# B&R Automation Studio project OpcUaSample410_BrbLibUa103 (part 16)

#### Set_BrbUaSrvGetMethodOperateText.c - Test set
```c
#include <bur/plctypes.h>

#ifdef _DEFAULT_INCLUDES
#include <AsDefault.h>
#endif

#include "UnitTest.h"
#include "BrbAsserts.h"
#include <string.h>

// NOLINTBEGIN(readability-*, bugprone-easily-swappable-parameters, bugprone-branch-clone, clang-diagnostic-invalid-utf8, clang-diagnostic-invalid-source-encoding, clang-diagnostic-pointer-arith, clang-diagnostic-strict-prototypes, clang-diagnostic-bad-function-cast, clang-analyzer-security.insecureAPI.*, hicpp-uppercase-literal-suffix, cppcoreguidelines-*, performance-*)
_TEST BrbUaSrvGetMethodOperateText_NulPtr(void)
{
	dwordOut = BrbUaSrvGetMethodOperateText(0, 0, 0);
	TEST_ASSERT_EQUAL_INT(0x80460000, dwordOut); // = Bad_StructureMissing

	// Finished
	TEST_DONE;
}

_TEST BrbUaSrvGetMethodOperateText_Get(void)
{
	methodOperationAction = UaMoa_CheckIsCalled;
	dwordOut = BrbUaSrvGetMethodOperateText(methodOperationAction, stringIn0, sizeof(stringIn0));
	TEST_ASSERT_EQUAL_INT(0x00000000, dwordOut); // = Good
	TEST_ASSERT_EQUAL_STRING("CheckIsCalled", stringIn0);

	methodOperationAction = UaMoa_Finished;
	dwordOut = BrbUaSrvGetMethodOperateText(methodOperationAction, stringIn0, sizeof(stringIn0));
	TEST_ASSERT_EQUAL_INT(0x00000000, dwordOut); // = Good
	TEST_ASSERT_EQUAL_STRING("Finished", stringIn0);

	// Finished
	TEST_DONE;
}

// NOLINTEND(readability-*, bugprone-easily-swappable-parameters, bugprone-branch-clone, clang-diagnostic-invalid-utf8, clang-diagnostic-invalid-source-encoding, clang-diagnostic-pointer-arith, clang-diagnostic-strict-prototypes, clang-diagnostic-bad-function-cast, clang-analyzer-security.insecureAPI.*, hicpp-uppercase-literal-suffix, cppcoreguidelines-*, performance-*)

/*
B+R UnitTest: This is generated code.
Do not edit! Do not move!
Description: UnitTest Testprogramm infrastructure (TestSet).
LastUpdated: 2023-04-25 13:44:36Z
By B+R UnitTest Helper Version: 2.0.1.59
*/
UNITTEST_FIXTURES(fixtures)
{
	new_TestFixture("BrbUaSrvGetMethodOperateText_NulPtr", BrbUaSrvGetMethodOperateText_NulPtr),
	new_TestFixture("BrbUaSrvGetMethodOperateText_Get", BrbUaSrvGetMethodOperateText_Get),
};

UNITTEST_CALLER_COMPLETE_EXPLICIT(Set_BrbUaSrvGetMethodOperateText, "Set_BrbUaSrvGetMethodOperateText", 0, 0, fixtures, 0, 0, 0);
```

### Package Logical/Tasks/Template - Muster für einen Task

### ReadMe.txt
```
Das ist nur ein Muster, um damit schnell die Grund-Struktur eines neuen Tasks zu erstellen.
Es wird für das Beispiel nicht benötigt.
```

### Program Logical/Tasks/Template/TemplateC/TemplateC (ANSIC) - Muster für einen C-Task

#### TemplateC.c - Implementation code
```c
#include <bur/plctypes.h>

#ifdef _DEFAULT_INCLUDES
	#include <AsDefault.h>
#endif

// NOLINTBEGIN(readability-*, bugprone-easily-swappable-parameters, bugprone-branch-clone, clang-diagnostic-invalid-utf8, clang-diagnostic-invalid-source-encoding, clang-diagnostic-pointer-arith, clang-diagnostic-strict-prototypes, clang-diagnostic-shadow, clang-diagnostic-bad-function-cast, clang-analyzer-security.insecureAPI.*, hicpp-uppercase-literal-suffix, hicpp-function-size, cppcoreguidelines-*, performance-*)

void _INIT Init(void)
{
}

void _CYCLIC Cyclic(void)
{
}

void _EXIT Exit(void)
{
}

// NOLINTEND(readability-*, bugprone-easily-swappable-parameters, bugprone-branch-clone, clang-diagnostic-invalid-utf8, clang-diagnostic-invalid-source-encoding, clang-diagnostic-pointer-arith, clang-diagnostic-strict-prototypes, clang-diagnostic-shadow, clang-diagnostic-bad-function-cast, clang-analyzer-security.insecureAPI.*, hicpp-uppercase-literal-suffix, hicpp-function-size, cppcoreguidelines-*, performance-*)
```

### Program Logical/Tasks/Template/TemplateST/TemplateST (IEC) - Muster für einen ST-Task

#### TemplateST.st - Init, cyclic, exit code
```iecst
PROGRAM _INIT
END_PROGRAM

PROGRAM _CYCLIC
END_PROGRAM

PROGRAM _EXIT
END_PROGRAM
```

### Package Logical/Tasks/ServerData - Daten für den eigenen OpcUa-Server

### ReadMe.txt
```
Hier werden Variablen zur Verfügung gestellt, die der eigene OpcUa-Server veröffentlicht.

Der Server ist in der System-Konfiguration unter 'OPCUA Server' parametriert. Es ist das PV-Informationsmodell V2.0
eingestellt.

Die User-/Roles-Parametrierung ist unter ConfigurationView/AccessAndSecurity/UserRoleSystem.  Hier ist folgende
Authentifizierung angegeben:
	Username:			Admin
	Password:			admin

Daten sind als globale Variable 'gVarsGlobal' und als lokale Variable 'VarsLocal' angelegt.
Sie wurden in der Datei 'OpcUaMap.uad' (siehe ConfigurationView/Connectivity/OpcUa) für den Server konfiguriert.
Sie enthalten die Strukturen 'Read', 'Write' und 'ReadWrite', welche auch so parametriert sind.
Diese wiederum enthalten jeweils ein Unterelement jeden Standard-Datentyps.
Definition siehe LogicalView/Global.typ.
Die Elemente der Unter-Struktur 'Read' werden im Task-Takt (500ms) geändert.

Eine Übersetzung des Attributes 'Description' ist beispielhaft bei den beiden Knoten 'gVarsGlobal' und 'VarsLocal'
implementiert. Dabei werden die Texte aus der Datei 'Texts/OpcUaServerTexts' verwendet.

Ausserdem gibt es die Strukturen 'WriteC' und 'WriteST', auf deren Elemente teilweise von den Clients geschrieben wird.

Einsatz von dynamischen Arrays:
	Auf einer SPS kann ein Array nie dynamisch sein, also keine variable Länge haben. Die Länge eines Arrays
	muss zur Projektierungszeit im AS  festgelegt werden und kann zur Laufzeit nicht mehr geändert werden.
	OpcUa untersützt jedoch dynamische Arrays.
	Der B&R-Server kann mit einem Trick ein in der SPS deklariertes Array OpcUa-seitig als dynamisch
	ausliefern. Auch ein empfangenes dynamisches Array kann so auf ein festes SPS-Array übertragen werden.
	Als einfaches Beispiel dient hier die Variable 'DynamicUintArrayLength', welche durch einen selbstdefinierten
	Datentyp deklariert wird. Der Datentyp sieht so aus:
		DynamicUintArrayLength_TYP : 	STRUCT
			nLength : UAArrayLength;
			anData : ARRAY[0..9]OF UINT;
		END_STRUCT;
	Das Element 'anData' enthält das Array mit fester maximaler Länge, wie auf der SPS benötigt.
	Das Element 'nLength' enthält die Anzahl der gültigen Array-Elemente. Durch Setzen dieses Wertes wird	das am
	OpcUa-Server bediente Array angepasst.
	Die Variable wird ganz normal am OpcUa-Server freigegeben (ohne Unter-Elemente). Das System erkennt aufgrund der
	Deklaration, dass diese	Variable ein dynamisches Array ist und behandelt es entsprechend.
	Bei einem DirectRead oder als MonitoredItem einer Subscription wird ein Array mit der aktuellen Länge übertragen.
	Bei einem DirectWrite werden die als Array übertragene Werte in 'anData' geschrieben und 'nLength' entsprechend
	gesetzt.
	Die Länge kann anstatt als 'UAArrayLength' auch als 'UANoOfElements' deklariert werden. Der Unterschied ist das Format,
	in welchem das Array an den Client übertragen bzw. vom Client erwartet wird:
		UAArrayLength:		Wird als Uint16[] übertragen.
		UANoOfElements:		Wird als ExtensionObject übertragen. Es enthält das UINT-Array.

	Als Beispiel für die zweite Variante ist die Variable 'DynamicUintArrayElements' implementiert. Über einen Test-Client
	wie UaExpert oder RnCommTest kann der Unterschied des Formats sehr leicht erkannt werden.
	Welche Variante verwendet werden sollte, hängt davon ab, mit welchem Format der Client umgehen kann. Sps-seitig ist
	Behandlung identisch.

	Dieses Konzept funktioniert nicht nur mit allen Standard-Datentypen, sondern auch mit Struktur-Arrays. Als Beispiele
	sind die beiden Variablen 'DynamicStructArrayLength' bzw. 'DynamicStructArrayElements' implementiert.
	Achtung: Mindestens eine skalare Instanz der verwendeten Struktur muss freigegeben sein, damit der Datentyp vom Server
	veröffentlicht wird und es dem Client so ermöglicht, die Struktur aufzulösen. Wenn der Struktur-Datentyp nur im Array
	verwendet wird, ist dies nicht der Fall!

	Achtung: Bei einem Schreib-Zugriff auf ein dynamisches Array darf die Anzahl der geschriebenen Elemente NICHT die
	Länge des Array 'anData' überschreiten, da der Server dann die empfangenen Daten nicht in das Array übertragen kann.
	Wird dies	doch gemacht, führt der Server den Schreibauftrag nicht aus und gibt den Status
	'0x8074000' = BadTypeMismatch	zurück!

	Hinweis: Bei dynamischen Arrays werden nur 1-dimensionale, aber keine mehrdimensionalen Arrays unterstützt.

	Implementierung im Beispiel-Task:
	Die Arrays werden im Init des Tasks vorbesetzt. Im zyklischen Teil (500ms) werden nur die Längen der einzelnen
	Instanzen zufällig verändert.

	Bekannte Bugs in AR-Versionen:
	Behoben ab C4.72:
		Definition mit 'UAArrayLength':
			Bei einem dynamischen Standard-Datentypen-Array, welches vom Client über eine	Subscription abonniert wurde,
			lieferte der Server bei einer Wert-Änderung nicht das Array, sondern nur die aktuelle Länge.
			Hinweis: Mit 'UANoOfElements' funktionierte es korrekt.

	Behoben ab B4.73:
		Definition mit 'UAArrayLength':
			Die Verwendung als Methoden-Argument funktioniert nicht korrekt. Werden weniger Elemente als die maximale Anzahl
			an Elementen gesendet, quittiert dies der Server mit '0x80AB000 = BadInvalidArgument'
			Hinweis: Mit 'UANoOfElements' funktioniert es korrekt.

Schreibbare Attribute:
	Die Variable 'nWritableAttributes' ist in der Datei 'OpcUaMap.uad' so parametriert, dass die Attribute
	'BrowseName', 'DisplayName' und 'Description' von einem Client beschrieben werden können.
	Achtung: Geänderte Werte sind nicht warmstartsicher!
```

### G_ServerData.var - Package variables
```iecst
VAR
	gVarsGlobal : OpcUaServerVars_TYP;
END_VAR
```

### Program Logical/Tasks/ServerData/ServerData (ANSIC) - Daten für den eigenen OpcUa-Server

#### ServerData.c - Implementation code
```c
#include <bur/plctypes.h>

#ifdef _DEFAULT_INCLUDES
	#include <AsDefault.h>
#endif

// NOLINTBEGIN(readability-*, bugprone-easily-swappable-parameters, bugprone-branch-clone, clang-diagnostic-invalid-utf8, clang-diagnostic-invalid-source-encoding, clang-diagnostic-pointer-arith, clang-diagnostic-strict-prototypes, clang-diagnostic-shadow, clang-diagnostic-bad-function-cast, clang-analyzer-security.insecureAPI.*, hicpp-uppercase-literal-suffix, hicpp-function-size, cppcoreguidelines-*, performance-*)

// Prototypen der lokalen Funktionen
void IncrementOpcUaTestDatatypes(OpcUaTestDatatypes_TYP* pDatatypes);
void ChangeDynamicArrays();

void _INIT Init(void)
{
	// Setzen der Test-Variablen
	brsmemset((UDINT)&gVarsGlobal, 0, sizeof(gVarsGlobal));
	brsstrcpy((UDINT)&gVarsGlobal.ReadOnly.sString, (UDINT)&"000");

	brsmemset((UDINT)&VarsLocal, 0, sizeof(VarsLocal));
	brsstrcpy((UDINT)&VarsLocal.ReadOnly.sString, (UDINT)&"000");

	brsmemset((UDINT)&WriteC, 0, sizeof(WriteC));
	brsmemset((UDINT)&WriteST, 0, sizeof(WriteST));

	// Diese Instanz der in den dynamischen Arrays verwendeten Struktur wird am Server freigegeben, damit dieser die Struktur-Definition veröffentlicht. Nur so kann ein Client diesen
	// benutzerdefinierten Datentypen auflösen.
	DummyStruct.nUsint = 0;

	DynamicUintArrayLength.nLength = 1;
	for(nIndex=0;nIndex<=nDYNAMIC_ARRAY_INDEX_MAX;nIndex++)
	{
		DynamicUintArrayLength.anData[nIndex] = nIndex;
	}
	DynamicUintArrayElements.nLength = 1;
	for(nIndex=0;nIndex<=nDYNAMIC_ARRAY_INDEX_MAX;nIndex++)
	{
		DynamicUintArrayElements.anData[nIndex] = nIndex;
	}
	DynamicStructArrayLength.nLength = 1;
	for(nIndex=0;nIndex<=nDYNAMIC_ARRAY_INDEX_MAX;nIndex++)
	{
		DynamicStructArrayLength.Data[nIndex].nUsint = (USINT)nIndex;
		DynamicStructArrayLength.Data[nIndex].rReal  = (REAL)nIndex + 0.1f;
	}
	DynamicStructArrayElements.nLength = 1;
	for(nIndex=0;nIndex<=nDYNAMIC_ARRAY_INDEX_MAX;nIndex++)
	{
		DynamicStructArrayElements.Data[nIndex].nUsint = (USINT)nIndex;
		DynamicStructArrayElements.Data[nIndex].rReal  = (REAL)nIndex + 0.1f;
	}

	nWritableAttributes = 123;
}

void _CYCLIC Cyclic(void)
{
	IncrementOpcUaTestDatatypes(&gVarsGlobal.ReadOnly);
	IncrementOpcUaTestDatatypes(&VarsLocal.ReadOnly);
	ChangeDynamicArrays();
}

void _EXIT Exit(void)
{
}

void IncrementOpcUaTestDatatypes(OpcUaTestDatatypes_TYP* pDatatypes)
{
	UINT		nStringLen;
	STRING	sHelpString[nOPCUA_STRING_CHAR_MAX];
	UINT		nHelpStringLen;

	pDatatypes->bBool = !pDatatypes->bBool;
	pDatatypes->nSint++;
	pDatatypes->nInt++;
	pDatatypes->nDint++;
	pDatatypes->nUsint++;
	pDatatypes->nUint++;
	pDatatypes->nUdint++;
	pDatatypes->rReal += 0.1f;
	pDatatypes->rLongReal += 0.2;
	pDatatypes->tTime++;
	pDatatypes->dtDateTime++;
	pDatatypes->anInt[0]++;
	pDatatypes->anInt[1]++;
	pDatatypes->anInt[2]++;
	pDatatypes->anInt[3]++;
	pDatatypes->anInt[4]++;

	nStringLen = (UINT)brsstrlen((UDINT)&pDatatypes->sString);
	brsitoa((DINT)pDatatypes->nUsint, (UDINT)&sHelpString);
	nHelpStringLen = (UINT)brsstrlen((UDINT)&sHelpString);
	if((nStringLen >= 3))
	{
		if(nHelpStringLen >= 3)
		{
			pDatatypes->sString[0] = sHelpString[0];
			pDatatypes->sString[1] = sHelpString[1];
			pDatatypes->sString[2] = sHelpString[2];
		}
		else if(nHelpStringLen == 2)
		{
			pDatatypes->sString[0] = 48;
			pDatatypes->sString[1] = sHelpString[0];
			pDatatypes->sString[2] = sHelpString[1];
		}
		else
		{
			pDatatypes->sString[0] = 48;
			pDatatypes->sString[1] = 48;
			pDatatypes->sString[2] = sHelpString[0];
		}
	}
	else if(nStringLen == 2)
	{
		if(nHelpStringLen >= 3)
		{
			pDatatypes->sString[0] = sHelpString[1];
			pDatatypes->sString[1] = sHelpString[2];
		}
		else if(nHelpStringLen == 2)
		{
			pDatatypes->sString[0] = sHelpString[0];
			pDatatypes->sString[1] = sHelpString[1];
		}
		else
		{
			pDatatypes->sString[0] = 48;
			pDatatypes->sString[1] = sHelpString[0];
		}
	}
	else if(nStringLen == 1)
	{
		if(nHelpStringLen >= 3)
		{
			pDatatypes->sString[0] = sHelpString[2];
		}
		else if(nHelpStringLen == 2)
		{
			pDatatypes->sString[0] = sHelpString[1];
		}
		else
		{
			pDatatypes->sString[0] = sHelpString[0];
		}
	}
}

void ChangeDynamicArrays()
{
	DynamicUintArrayLength.nLength = BrbGetRandomDint(1, 5);
	DynamicUintArrayElements.nLength = BrbGetRandomDint(1, 5);
	DynamicStructArrayLength.nLength = BrbGetRandomDint(1, 5);
	DynamicStructArrayElements.nLength = BrbGetRandomDint(1, 5);
}

// NOLINTEND(readability-*, bugprone-easily-swappable-parameters, bugprone-branch-clone, clang-diagnostic-invalid-utf8, clang-diagnostic-invalid-source-encoding, clang-diagnostic-pointer-arith, clang-diagnostic-strict-prototypes, clang-diagnostic-shadow, clang-diagnostic-bad-function-cast, clang-analyzer-security.insecureAPI.*, hicpp-uppercase-literal-suffix, hicpp-function-size, cppcoreguidelines-*, performance-*)
```

#### ServerData.typ - Local data types
```iecst
TYPE
	DynamicUintArrayLength_TYP : 	STRUCT
		nLength : UAArrayLength;
		anData : ARRAY[0..9]OF UINT; (*nDYNAMIC_ARRAY_INDEX_MAX*)
	END_STRUCT;
	DynamicUintArrayElements_TYP : 	STRUCT
		nLength : UANoOfElements;
		anData : ARRAY[0..9]OF UINT; (*nDYNAMIC_ARRAY_INDEX_MAX*)
	END_STRUCT;
	OpcUaTest_TYP : 	STRUCT
		nUsint : USINT;
		rReal : REAL;
	END_STRUCT;
	DynamicStructArrayLength_TYP : 	STRUCT
		nLength : UAArrayLength;
		Data : ARRAY[0..9]OF OpcUaTest_TYP; (*nDYNAMIC_ARRAY_INDEX_MAX*)
	END_STRUCT;
	DynamicStructArrayElements_TYP : 	STRUCT
		nLength : UANoOfElements;
		Data : ARRAY[0..9]OF OpcUaTest_TYP; (*nDYNAMIC_ARRAY_INDEX_MAX*)
	END_STRUCT;
END_TYPE
```

#### ServerData.var - Local variables
```iecst
VAR
	VarsLocal : OpcUaServerVars_TYP;
	WriteC : OpcUaTestDatatypes_TYP;
	WriteST : OpcUaTestDatatypes_TYP;
	nIndex : UINT;
END_VAR
VAR CONSTANT
	nDYNAMIC_ARRAY_INDEX_MAX : UINT := 9;
END_VAR
VAR
	DummyStruct : OpcUaTest_TYP;
	DynamicUintArrayLength : DynamicUintArrayLength_TYP;
	DynamicUintArrayElements : DynamicUintArrayElements_TYP;
	DynamicStructArrayLength : DynamicStructArrayLength_TYP;
	DynamicStructArrayElements : DynamicStructArrayElements_TYP;
	nWritableAttributes : USINT;
END_VAR
```

### Package Logical/Tasks/ServerDt64 - Behandlung von 64-Bit-Datentypen

### ReadMe.txt
```
Die größten nativ auf der Sps unter IEC unterstützten Integer-Datentypen sind UDINT (Uint32) und DINT (Int32).
Manchmal werden aber auch größere Datentypen als Zähler benötigt (z.B. bei Companion Specifications).

Dieses Beispiel zeigt die Verwendung von 64-Bit-Datentypen wie Uint64 (ULINT) und Int64 (LINT) unter OpcUa.
Die benötigten Strukturen und Funktionen dafür sind in der Basis-Bibliothek BrbLib ab V5.02 implementiert.
Beschreibungen und Hinweise dazu sind in der Hilfe der Bibliothek zu finden. Besonders beachtet werden sollte
der Hinweis zur Konsistenz!

Der Task definiert jeweils einen Uint64 (Variable nUint64) und einen Int64 (Variable nInt64).
Beide werden zyklisch verändert, um den Umgang damit zu demonstrieren. Vor allem die Unter- bzw. Überläufe
werden dabei gezeigt:

	Uint64:
		Bereich: 0..18446744073709551615
		Startwert: 0
		Er wird auf 5 hochgezählt. Dann wird die Zählrichtung auf negativ gesetzt. Wird er bei 0 (=niedrigster Wert)
		nochmals um 1 dekrementiert, findet ein Unterlauf statt, der zum Wert 18446744073709551615 (=höchster Wert) führt.
		Es wird dann weiter bis 18446744073709551610 runtergezählt. Dann wird die Zählrichtung wieder auf positiv gesetzt.
		Wird bei 18446744073709551615 (=höchster Wert) nochmals um 1 inkrementiert, findet ein Überlauf statt, der zum Wert
		0 (=niedrigster Wert) führt. Dann startet die Zählung von vorne.
		Die Unter- bzw. Überlauf-Logik ist also gleich wie bei einem vorzeichenlosen Wert mit weniger Bits (z.B. ein UINT).
		Um den 64-Bit-Wert auf der Sps menschenlesbar zu machen, wird er zyklisch in einen Text gewandelt, der die tatsächliche
		Zahl zeigt (Variable sUint64).

	Int64:
		Bereich: -9223372036854775808..+9223372036854775807
		Startwert: +9223372036854775802
		Er wird auf +9223372036854775807 (=höchster Wert) hochgezählt. Wird dann nochmals um 1 inkrementiert, findet ein
		Überlauf statt, der zum Wert -9223372036854775808 (=niedrigster Wert) führt. Es wird weiter hochgezählt
		auf -9223372036854775803. Dann wird die Zählrichtung auf negativ gesetzt. Wird beim Wert -9223372036854775808
		(=niedrigster Wert) nochmals um 1 dekrementiert, findet ein Unterlauf statt, der zum Wert +9223372036854775807
		(=höchster Wert) führt. Es wird weiter runtergezählt bis +9223372036854775802 und dann die Zählrichtung wieder auf
		positiv gesetzt. Dann startet die Zählung von vorne.
		Die Unter- bzw. Überlauf-Logik ist also gleich wie bei einem vorzeichenbehafteten Wert mit weniger Bits (z.B.
		ein INT).
		Um den 64-Bit-Wert auf der Sps menschenlesbar zu machen, wird er zyklisch in einen Text gewandelt, der die tatsächliche
		Zahl zeigt (Variable sInt64).

Veröffentlichung am OpcUa-Server als 64-Bit-Wert:
	Auf der Sps sind die 64-Bit-Werte also als Struktur aufgelegt (BrbUint64_TYP bzw. BrbInt64_TYP).
	Um den Server dazu zu bringen, diese Struktur als Uint64 bzw. Int64 zu veröffentlichen, ist nur eine einfache
	Konfiguration nötig. Sie muss in der Datei 'OpcUaMap.uad' (siehe ConfigurationView/Connectivity/OpcUa) gemacht werden,
	und zwar in der Spalte 'UA Datatype' der Struktur-Variable (die Unterelemente der Struktur sollten nicht freigegeben
	werden). Hier kann optional ein anderer als der Sps-Datentyp als NodeId des OpcUa-Datentyps angegeben werden:
		Uint64: ns=0;i=9
		Int64: ns=0;i=8
	Der Server veröffentlicht dann den Variablen-Wert als angegebenen OpcUa-Datentyp.
	Dies funktioniert aber nur, wenn die Sps-Variable die Länge in Bytes hat, welche vom angegebenen OpcUa-Typ benötigt wird.
	Die OpcUa-Datentypen Uint64 bzw. Int64 benötigen jeweils 8 Byte, welche durch die Instanzen der Strukturen
	'BrbUint64_TYP' bzw. 'BrbInt64_TYP' bereitgestellt werden.
```

### Program Logical/Tasks/ServerDt64/SrvDt64C/SrvDt64C (ANSIC) - Behandlung von 64-Bit-Datentypen in ANSI-C

#### SrvDt64C.c - Implementation code
```c
#include <bur/plctypes.h>

#ifdef _DEFAULT_INCLUDES
	#include <AsDefault.h>
#endif

// NOLINTBEGIN(readability-*, bugprone-easily-swappable-parameters, bugprone-branch-clone, clang-diagnostic-invalid-utf8, clang-diagnostic-invalid-source-encoding, clang-diagnostic-pointer-arith, clang-diagnostic-strict-prototypes, clang-diagnostic-shadow, clang-diagnostic-bad-function-cast, clang-analyzer-security.insecureAPI.*, hicpp-uppercase-literal-suffix, hicpp-function-size, cppcoreguidelines-*, performance-*)

// Prototypen der lokalen Funktionen
void ChangeUint64();
void ChangeInt64();

void _INIT Init(void)
{
	// Uint64 und Zähler-Grenzen setzen
	BrbUint64FromString(&nUint64, "0");
	BrbUint64FromString(&ChangeUint64Inst.nCountMin, "5");
	BrbUint64FromString(&ChangeUint64Inst.nCountMax, "18446744073709551610");
	ChangeUint64Inst.bCountPositive = 1;

	// Int64 und Zähler-Grenzen setzen
	BrbInt64FromString(&nInt64, "9223372036854775802");
	BrbInt64FromString(&ChangeInt64Inst.nCountMin, "-9223372036854775803");
	BrbInt64FromString(&ChangeInt64Inst.nCountMax, "9223372036854775802");
	ChangeInt64Inst.bCountPositive = 1;
}

void _CYCLIC Cyclic(void)
{
	ChangeUint64(); // Wert zyklisch ändern
	BrbUint64ToString(&nUint64, sUint64, sizeof(sUint64)); // In Text für bessere Lesbarkeit wandeln

	ChangeInt64(); // Wert zyklisch ändern
	BrbInt64ToString(&nInt64, sInt64, sizeof(sInt64)); // In Text für bessere Lesbarkeit wandeln
}

void _EXIT Exit(void)
{
}

// Ändern des Uint64-Wertes
void ChangeUint64()
{
	if(ChangeUint64Inst.bCountPositive == 1)
	{
		BrbUint64Inc(&nUint64);
		if(BrbUint64Compare(&nUint64, &ChangeUint64Inst.nCountMin) == 0)
		{
			ChangeUint64Inst.bCountPositive = 0;
		}
	}
	else
	{
		BrbUint64Dec(&nUint64);
		if(BrbUint64Compare(&nUint64, &ChangeUint64Inst.nCountMax) == 0)
		{
			ChangeUint64Inst.bCountPositive = 1;
		}
	}
}

// Ändern des Int64-Wertes
void ChangeInt64()
{
	if(ChangeInt64Inst.bCountPositive == 1)
	{
		BrbInt64Inc(&nInt64);
		if(BrbInt64Compare(&nInt64, &ChangeInt64Inst.nCountMin) == 0)
		{
			ChangeInt64Inst.bCountPositive = 0;
		}
	}
	else
	{
		BrbInt64Dec(&nInt64);
		if(BrbInt64Compare(&nInt64, &ChangeInt64Inst.nCountMax) == 0)
		{
			ChangeInt64Inst.bCountPositive = 1;
		}
	}
}

// NOLINTEND(readability-*, bugprone-easily-swappable-parameters, bugprone-branch-clone, clang-diagnostic-invalid-utf8, clang-diagnostic-invalid-source-encoding, clang-diagnostic-pointer-arith, clang-diagnostic-strict-prototypes, clang-diagnostic-shadow, clang-diagnostic-bad-function-cast, clang-analyzer-security.insecureAPI.*, hicpp-uppercase-literal-suffix, hicpp-function-size, cppcoreguidelines-*, performance-*)
```

#### SrvDt64C.typ - Local data types
```iecst
TYPE
	ChangeUint64C_TYP : 	STRUCT
		bCountPositive : BOOL;
		nCountMin : BrbUint64_TYP;
		nCountMax : BrbUint64_TYP;
	END_STRUCT;
	ChangeInt64C_TYP : 	STRUCT
		bCountPositive : BOOL;
		nCountMin : BrbInt64_TYP;
		nCountMax : BrbInt64_TYP;
	END_STRUCT;
END_TYPE
```

#### SrvDt64C.var - Local variables
```iecst
VAR
	nUint64 : BrbUint64_TYP;
	sUint64 : STRING[nBRB_UINT64_CHAR_MAX];
	ChangeUint64Inst : ChangeUint64C_TYP;
	nInt64 : BrbInt64_TYP;
	sInt64 : STRING[nBRB_INT64_CHAR_MAX];
	ChangeInt64Inst : ChangeInt64C_TYP;
END_VAR
```

### Program Logical/Tasks/ServerDt64/ServerDt64ST/SrvDt64ST (IEC) - Behandlung von 64-Bit-Datentypen in ST

#### SrvDt64ST.st - Init, cyclic, exit code
```iecst
PROGRAM _INIT
	// Uint64 und Zähler-Grenzen setzen
	pUint64 ACCESS ADR(nUint64);
	BrbUint64FromString(pUint64, '0');
	pUint64CountMin ACCESS ADR(ChangeUint64Inst.nCountMin);
	BrbUint64FromString(pUint64CountMin, '5');
	pUint64CountMax ACCESS ADR(ChangeUint64Inst.nCountMax);
	BrbUint64FromString(pUint64CountMax, '18446744073709551610');
	ChangeUint64Inst.bCountPositive := 1;

	// Int64 und Zähler-Grenzen setzen
	pInt64 ACCESS ADR(nInt64);
	BrbInt64FromString(pInt64, '9223372036854775802');
	pInt64CountMin ACCESS ADR(ChangeInt64Inst.nCountMin);
	BrbInt64FromString(pInt64CountMin, '-9223372036854775803');
	pInt64CountMax ACCESS ADR(ChangeInt64Inst.nCountMax);
	BrbInt64FromString(pInt64CountMax, '9223372036854775802');
	ChangeInt64Inst.bCountPositive := 1;
END_PROGRAM

PROGRAM _CYCLIC
	ChangeUint64; // Wert zyklisch ändern
	BrbUint64ToString(pUint64, sUint64, SIZEOF(sUint64)); // In Text für bessere Lesbarkeit wandeln

	ChangeInt64; // Wert zyklisch ändern
	BrbInt64ToString(pInt64, sInt64, SIZEOF(sInt64)); // In Text für bessere Lesbarkeit wandeln
END_PROGRAM

PROGRAM _EXIT
END_PROGRAM
```

#### SrvDt64ST.typ - Local data types
```iecst
TYPE
	ChangeUint64ST_TYP : 	STRUCT
		bCountPositive : BOOL;
		nCountMin : BrbUint64_TYP;
		nCountMax : BrbUint64_TYP;
	END_STRUCT;
	ChangeInt64ST_TYP : 	STRUCT
		bCountPositive : BOOL;
		nCountMin : BrbInt64_TYP;
		nCountMax : BrbInt64_TYP;
	END_STRUCT;
END_TYPE
```

#### SrvDt64ST.var - Local variables
```iecst
VAR
	nUint64 : BrbUint64_TYP;
	sUint64 : STRING[nBRB_UINT64_CHAR_MAX];
	pUint64 : REFERENCE TO BrbUint64_TYP;
	pUint64CountMin : REFERENCE TO BrbUint64_TYP;
	pUint64CountMax : REFERENCE TO BrbUint64_TYP;
	ChangeUint64Inst : ChangeUint64ST_TYP;
	nInt64 : BrbInt64_TYP;
	sInt64 : STRING[nBRB_INT64_CHAR_MAX];
	pInt64 : REFERENCE TO BrbInt64_TYP;
	pInt64CountMin : REFERENCE TO BrbInt64_TYP;
	pInt64CountMax : REFERENCE TO BrbInt64_TYP;
	ChangeInt64Inst : ChangeInt64ST_TYP;
END_VAR
```

#### Action.st
```iecst
// Ändern des Uint64-Wertes
ACTION ChangeUint64:
	IF ChangeUint64Inst.bCountPositive = 1 THEN
		BrbUint64Inc(pUint64);
		IF BrbUint64Compare(pUint64, pUint64CountMin) = 0 THEN
			ChangeUint64Inst.bCountPositive := 0;
		END_IF
	ELSE
		BrbUint64Dec(pUint64);
		IF BrbUint64Compare(pUint64, pUint64CountMax) = 0 THEN
			ChangeUint64Inst.bCountPositive := 1;
		END_IF
	END_IF
END_ACTION

// Ändern des Int64-Wertes
ACTION ChangeInt64:
	IF ChangeInt64Inst.bCountPositive = 1 THEN
		BrbInt64Inc(pInt64);
		IF BrbInt64Compare(pInt64, pInt64CountMin) = 0 THEN
			ChangeInt64Inst.bCountPositive := 0;
		END_IF
	ELSE
		BrbInt64Dec(pInt64);
		IF BrbInt64Compare(pInt64, pInt64CountMax) = 0 THEN
			ChangeInt64Inst.bCountPositive := 1;
		END_IF
	END_IF
END_ACTION
```

### Package Logical/Tasks/ServerMethods - Methoden-Aufruf im Server

### ReadMe.txt
```
Beispiel-Methode 'Calculate'
Die Methode ist in der Datei 'Methods.uam' deklariert, welche zum Task hinzugefügt wurde.
Sie enthält 3 Eingangs-Argumente ('nValue0', 'nValue1' und 'anArrayIn') sowie 3 Ausgangs-
Argumente ('nAddition', 'nMultiplication' und 'anArrayOut').
Die Eingangswerte werden sowohl addiert als auch multipliziert. Das Array wird nur auf den Ausgang
übernommen.

Die Methode ist in der Datei 'OpcUaMap.uad' (siehe ConfigurationView/Connectivity/OpcUa) für den Server konfiguriert.

Ablauf:
	1. Es wird geprüft, ob die Methode von einem Client aufgerufen wurde. Wenn ja, wird auf 2. geprungen
	2. Der applikative Code der Methode wird ausgeführt (Addition, Multiplikation + Übernahme des Arrays)
	3. Es wird zurückgemeldet, dass die Methode ausgeführt wurde

Beim Aufruf werden die Eingangs-Argumente in der lokalen Struktur 'MethCalculateArgs.In' übergeben.
Die Ausgangs-Argumente können über die lokale Struktur 'MethCalculateArgs.Out' zurückgegeben werden.
```

### Package Logical/Tasks/ServerMethods/SrvMethC - Methoden-Aufruf im Server in ANSI-C

### Program Logical/Tasks/ServerMethods/SrvMethC/SrvMethC (ANSIC) - Methoden-Aufruf im Server in ANSI-C

#### SrvMethC.c - Implementation code
```c
#include <bur/plctypes.h>

#ifdef _DEFAULT_INCLUDES
	#include <AsDefault.h>
#endif

// NOLINTBEGIN(readability-*, bugprone-easily-swappable-parameters, bugprone-branch-clone, clang-diagnostic-invalid-utf8, clang-diagnostic-invalid-source-encoding, clang-diagnostic-pointer-arith, clang-diagnostic-strict-prototypes, clang-diagnostic-shadow, clang-diagnostic-bad-function-cast, clang-analyzer-security.insecureAPI.*, hicpp-uppercase-literal-suffix, hicpp-function-size, cppcoreguidelines-*, performance-*)

void _INIT Init(void)
{
	// Ablöschen der Funktionsblöcke und Strukturen
	brsmemset((UDINT)&fbUaSrv_MethodOperateCalculate, 0, sizeof(fbUaSrv_MethodOperateCalculate));
	brsmemset((UDINT)&MethCalculateArgs, 0, sizeof(MethCalculateArgs));

	// Setzen der Methode 'Calculate'
	brsstrcpy((UDINT)&fbUaSrv_MethodOperateCalculate.MethodName, (UDINT)&"Calculate"); // Name der Methode wie in 'Methods.uam' angegeben

	// Initialisierung der Schrittkette
	Step.eStepNr = eSTEP_CHECK;

}

void _CYCLIC Cyclic(void)
{

	// Schrittkette
	switch(Step.eStepNr)
	{
		case eSTEP_NONE:

		case eSTEP_CHECK:
			// Prüfen, ob Methode von einem Client aufgerufen wurde
			fbUaSrv_MethodOperateCalculate.Execute = 1;
			fbUaSrv_MethodOperateCalculate.Action = UaMoa_CheckIsCalled;
			if(fbUaSrv_MethodOperateCalculate.Done == 1)
			{
				fbUaSrv_MethodOperateCalculate.Execute = 0;
				if(fbUaSrv_MethodOperateCalculate.IsCalled == 1)
				{
					// Variablen der Eingans-Argumente sind besetzt -> Methode ausführen
					Step.eStepNr = eSTEP_EXECUTE;
				}
			}
			else if(fbUaSrv_MethodOperateCalculate.Error == 1)
			{
				fbUaSrv_MethodOperateCalculate.Execute = 0;
				Step.eErrorStep = Step.eStepNr;
				Step.eAction = fbUaSrv_MethodOperateCalculate.Action;
				Step.nErrorId = fbUaSrv_MethodOperateCalculate.ErrorID;
			}
			break;

		case eSTEP_EXECUTE:
			// Ausführen der Methode (Besetzen der Ausgangs-Argumente)
			MethCalculateArgs.Out.nAddition = MethCalculateArgs.In.nVal0 + MethCalculateArgs.In.nVal1;
			MethCalculateArgs.Out.nMultiplication = MethCalculateArgs.In.nVal0 * MethCalculateArgs.In.nVal1;
			brsmemcpy((UDINT)&MethCalculateArgs.Out.anArray, (UDINT)&MethCalculateArgs.In.anArray, sizeof(MethCalculateArgs.Out.anArray)); // In-Array auf Out-Array übernehmen

			nMethCalculateCallCount += 1; // Nur zur Diagnose
			Step.eStepNr = eSTEP_FINSHED;
			break;

		case eSTEP_FINSHED:
			// Rückmelden, dass Methode ausgeführt wurde. Zu diesem Zeitpunkt müssen die Ausgangs-Argumente besetzt sein und dürfen nicht mehr geändert werden
			fbUaSrv_MethodOperateCalculate.Execute = 1;
			fbUaSrv_MethodOperateCalculate.Action = UaMoa_Finished;
			if(fbUaSrv_MethodOperateCalculate.Done == 1)
			{
				fbUaSrv_MethodOperateCalculate.Execute = 0;
				Step.eStepNr = eSTEP_CHECK;
			}
			else if(fbUaSrv_MethodOperateCalculate.Error == 1)
			{
				// Fehler eintragen, aber trotzdem weiter machen
				fbUaSrv_MethodOperateCalculate.Execute = 0;
				Step.eErrorStep = Step.eStepNr;
				Step.eAction = fbUaSrv_MethodOperateCalculate.Action;
				Step.nErrorId = fbUaSrv_MethodOperateCalculate.ErrorID;
				Step.eStepNr = eSTEP_CHECK;
			}
			break;

	}

	// Aufruf aller PlcOpen-Funktionsblöcke
	UaSrv_MethodOperate(&fbUaSrv_MethodOperateCalculate);
}

void _EXIT Exit(void)
{
}

// NOLINTEND(readability-*, bugprone-easily-swappable-parameters, bugprone-branch-clone, clang-diagnostic-invalid-utf8, clang-diagnostic-invalid-source-encoding, clang-diagnostic-pointer-arith, clang-diagnostic-strict-prototypes, clang-diagnostic-shadow, clang-diagnostic-bad-function-cast, clang-analyzer-security.insecureAPI.*, hicpp-uppercase-literal-suffix, hicpp-function-size, cppcoreguidelines-*, performance-*)
```

### Package Logical/Tasks/ServerMethods/SrvMethST - Methoden-Aufruf im Server In ST

### Program Logical/Tasks/ServerMethods/SrvMethST/SrvMethST (IEC) - Methoden-Aufruf im Server In ST

#### Main.st - Init, cyclic, exit code
```iecst
PROGRAM _INIT
	// Ablöschen der Funktionsblöcke und Strukturen
	brsmemset(ADR(fbUaSrv_MethodOperateCalculate), 0, SIZEOF(fbUaSrv_MethodOperateCalculate));
	brsmemset(ADR(MethCalculateArgs), 0, SIZEOF(MethCalculateArgs));

	// Setzen der Methode 'Calculate'
	fbUaSrv_MethodOperateCalculate.MethodName := 'Calculate'; // Name der Methode wie in 'Methods.uam' angegeben

	// Initialisierung der Schrittkette
	Step.eStepNr := eSTEP_CHECK;

END_PROGRAM

PROGRAM _CYCLIC

		// Schrittkette
	CASE Step.eStepNr OF
		eSTEP_NONE:

		eSTEP_CHECK:
			// Prüfen, ob Methode von einem Client aufgerufen wurde
			fbUaSrv_MethodOperateCalculate.Execute := 1;
			fbUaSrv_MethodOperateCalculate.Action := UaMoa_CheckIsCalled;
			IF fbUaSrv_MethodOperateCalculate.Done = 1 THEN
				fbUaSrv_MethodOperateCalculate.Execute := 0;
				IF fbUaSrv_MethodOperateCalculate.IsCalled = 1 THEN
					// Variablen der Eingans-Argumente sind besetzt -> Methode ausführen
					Step.eStepNr := eSTEP_EXECUTE;
				END_IF
			ELSIF fbUaSrv_MethodOperateCalculate.Error = 1 THEN
				fbUaSrv_MethodOperateCalculate.Execute := 0;
				Step.eErrorStep := Step.eStepNr;
				Step.eAction := fbUaSrv_MethodOperateCalculate.Action;
				Step.nErrorId := fbUaSrv_MethodOperateCalculate.ErrorID;
			END_IF

		eSTEP_EXECUTE:
			// Ausführen der Methode
			MethCalculateArgs.Out.nAddition := MethCalculateArgs.In.nVal0 + MethCalculateArgs.In.nVal1;
			MethCalculateArgs.Out.nMultiplication := MethCalculateArgs.In.nVal0 * MethCalculateArgs.In.nVal1;
			brsmemcpy(ADR(MethCalculateArgs.Out.anArray), ADR(MethCalculateArgs.In.anArray), SIZEOF(MethCalculateArgs.Out.anArray)); // In-Array auf Out-Array übernehmen

			nMethCalculateCallCount := nMethCalculateCallCount + 1; // Nur zur Diagnose
			Step.eStepNr := eSTEP_FINSHED;

		eSTEP_FINSHED:
			// Rückmelden, dass Methode ausgeführt wurde. Zu diesem Zeitpunkt müssen die Ausgangs-Argumente besetzt sein und dürfen nicht mehr geändert werden
			fbUaSrv_MethodOperateCalculate.Execute := 1;
			fbUaSrv_MethodOperateCalculate.Action := UaMoa_Finished;
			IF fbUaSrv_MethodOperateCalculate.Done = 1 THEN
				fbUaSrv_MethodOperateCalculate.Execute := 0;
				Step.eStepNr := eSTEP_CHECK;
			ELSIF fbUaSrv_MethodOperateCalculate.Error = 1 THEN
				// Fehler eintragen, aber trotzdem weiter machen
				fbUaSrv_MethodOperateCalculate.Execute := 0;
				Step.eErrorStep := Step.eStepNr;
				Step.eAction := fbUaSrv_MethodOperateCalculate.Action;
				Step.nErrorId := fbUaSrv_MethodOperateCalculate.ErrorID;
				Step.eStepNr := eSTEP_CHECK;
			END_IF

	END_CASE

	// Aufruf aller PlcOpen-Funktionsblöcke
	fbUaSrv_MethodOperateCalculate();

END_PROGRAM

PROGRAM _EXIT
END_PROGRAM
```

#### Types.typ - Local data types
```iecst
TYPE
	Step_TYP : 	STRUCT
		eStepNr : Steps_ENUM;
		eErrorStep : Steps_ENUM;
		eAction : UaMethodOperateAction;
		nErrorId : DWORD;
	END_STRUCT;
	Steps_ENUM :
		(
		eSTEP_NONE,
		eSTEP_CHECK,
		eSTEP_EXECUTE,
		eSTEP_FINSHED
		);
END_TYPE
```

#### Variables.var - Local variables
```iecst
VAR
	Step : Step_TYP;
	fbUaSrv_MethodOperateCalculate : UaSrv_MethodOperate;
	MethCalculateArgs : MethCalculateArgs_TYP;
	nMethCalculateCallCount : UDINT;
END_VAR
```

- Methods.uam (not shown)

### Package Logical/Tasks/ServerEvents - Event-Aufruf im Server

### ReadMe.txt
```
Beispiel zum anwenderseitigen Feuern eines Events.

Gefeuert wird in diesem Beispiel das Event 'ProgressEventType'. Es wird normalerweise dazu verwendet, den
Fortschritt eines Prozesses zu melden.
Da es direkt von 'BaseEventType' abgeleitet ist, besitzt es dessen Felder 'EventId', 'EventType', 'LocalTime',
'Message', 'ReceiveTime', 'Severity', 'SourceName', 'SourceNode' und 'Time'.
Im Task besetzt werden davon nur 'Message' und 'Severity'. Die anderen werden nicht übergeben und daher
automatisch vom Betriebssystem besetzt:
'EventId' enthält eine automatisch erstellte, eindeutige GUID.
'EventType' enthält 'ns=0;i=11436'. Das ist der Knoten von 'ProgressEventType'.
'LocalTime' enthält die Differenz der lokalen Server-Zeit zur UTC-Zeit.
'ReceiveTime' enthält die UTC-Zeit, wann das Event vom Server empfangen wurde, falls der Server nicht der Erzeuger
	des Events ist. In diesem Fall wird sie nicht besetzt und ist daher gleich 'Time'.
'SourceName' enthält den DisplayName des Knotens, der bei 'SourceNode' angegeben ist.
'SourceNode' enthält die NodeId des Knotens, der der Auslöser des Events ist. Da sie hier nicht applikativ besetzt wird,
	wird sie vom System automatisch als "i=0" besetzt.
'Time' enthält die UTC-Zeit, wann das Event aufgetreten ist.

Bei jedem Feuern werden anwenderseitig folgende BaseEvent-Felder besetzt:
'Message' sollte einen LocalizedText enthalten, welcher das Event durch einen Klartext beschreibt.
'Severity' sollte die Priorität des Events (1=Info; 1000=Katastrophe) enthalten. In diesem Beispiel wird er als
	Zufallszahl	zwischen 1 und 500 gebildet.

Das gefeuerte Event 'ProgressEventType' enthält aber auch noch die eigenen Felder 'Context' und 'Progress':
'Context' hat als Datentypen 'BaseDataType'. Damit ist es ein Variant und kann alle Datentypen aufnehmen.
	In diesem Beispiel wird der Wert in Form der benutzerdefinierten Struktur 'FieldContext_TYP' übergeben.
	Es wäre aber auch möglich, eine Variable vom Datentyp 'REAL' oder 'UDINT' usw. anzugeben.
	Achtung: Damit ein Client diese als ExtensionObject (Byte-Array) gesendete Struktur wieder auflösen kann,
	ist es unbedingt erforderlich, dass mindestens eine Instanz dieses Datentyps am Server freigegeben ist
	(siehe OpcUaMap.uad). Nur so veröffentlicht der Server automatisch die Definition dieser Struktur!
	Achtung: Fehler in einigen AR-Versionen (A4.90 bis D4.90)
		Leider liefert der FB den Fehler 0x803D0000 = 'Bad_NotSupported' zurück, wenn eine Struktur an diesem Feld
		angebunden ist, deren Typ-Defintion global angelegt ist. Ab E4.90 ist dieser Fehler behoben.
		Muss eine dieser fehlerhaften Versionen verwendet werden, so kann als Workaround die Definition der Struktur
		lokal gemacht werden.

'Progress' enthält den Wert des Fortschritts als UINT und wird in diesem Beispiel bei jedem Feuern hochgezählt.
	Der Fortschritt wird hier als % interpretiert und daher nach 100% also wieder auf 0 gesetzt.

Prinzipiell muss die an das Feld gebundene Variable dem Datentyp des Feldes entsprechen. Ist das Feld vom Datentyp
'BaseDataType' (Variant), so kann jeder Datentyp angebunden werden.

Ablauf der Schrittkette:
	eSTEP_INIT:								Start der Schrittkette
	eSTEP_GET_NS_ORG:					Ermitteln des NamespaceIndex für 'http://opcfoundation.org/UA/'
	eSTEP_GET_NS_BR_PV:				Ermitteln des NamespaceIndex für 'http://br-automation.com/OpcUa/PLC/PV/'
	eSTEP_DELAY:							Warten auf Timer
	eSTEP_SET_FIELD_VALUES:		Anwenderseitiges Besetzen der Event-Felder
	eSTEP_FIRE:								Feuern des Events

Die Namespace-Uris sind fest vergeben und ändern sich nicht. Die zugehörigen Namespace-Indizes werden beim Hochlauf
	des Servers vergeben und müssen daher ermittelt werden.
Durch einen Timer wird das Event jede 5 Sekunden gefeuert. Durch die Variable 'bSuspendTimer' kann dies verhindert
	werden. Durch die Variable 'bFire' kann das Event dann manuell gefeuert werden.

Um clientseitig das Event emfpangen zu können, muss der Knoten 'ns=0;i=2253' (Root/Objects/Server) in einer
Subscription abonniert werden. Ausserdem muss der Filter des EventItems die zu schickenden Felder enthalten.
Hinweis: Beim frei erhältlichen Test-Client 'UaExpert' ist beim Abonnieren des Knotens der Filter automatisch so
gesetzt, dass er alle Felder enthält.
Bei anderen Test-Client (z.B. RnCommTest) können der Filter und damit die Felder evtl. parametriert werden.
Im Task 'Client' ist ein Beispiel enthalten, wie auf der Sps dieses Event empfangen werden kann.

Da sowohl der ANSIC-Task als auch der ST-Task unabhängig voneinander arbeiten, würde das Event immer von beiden Tasks
gefeuert. Aus diesem Grund sollte immer einer der Tasks disabled sein. Hier ist es der Task 'SrvEvntST'.
```

### Package Logical/Tasks/ServerEvents/SrvEvntC - Event-Aufruf im Server in ANSI-C

### Program Logical/Tasks/ServerEvents/SrvEvntC/SrvEvntC (ANSIC) - Event-Aufruf im Server in ANSI-C

#### SrvEvntC.c - Implementation code
```c
#include <bur/plctypes.h>

#ifdef _DEFAULT_INCLUDES
	#include <AsDefault.h>
#endif

// NOLINTBEGIN(readability-*, bugprone-easily-swappable-parameters, bugprone-branch-clone, clang-diagnostic-invalid-utf8, clang-diagnostic-invalid-source-encoding, clang-diagnostic-pointer-arith, clang-diagnostic-strict-prototypes, clang-diagnostic-shadow, clang-diagnostic-bad-function-cast, clang-analyzer-security.insecureAPI.*, hicpp-uppercase-literal-suffix, hicpp-function-size, cppcoreguidelines-*, performance-*)

void _INIT Init(void)
{
	// Ablöschen der Funktionsblöcke und Strukturen
	brsmemset((UDINT)&fbUaSrv_GetNamespaceIndex, 0, sizeof(fbUaSrv_GetNamespaceIndex));
	brsmemset((UDINT)&fbUaSrv_FireEvent, 0, sizeof(fbUaSrv_FireEvent));
	brsmemset((UDINT)&Fields, 0, sizeof(Fields));

	// Setzen des Events 'ProgressEventType'
	fbUaSrv_FireEvent.EventType.NamespaceIndex = 0; // Wird in der Schrittkette ermittelt
	fbUaSrv_FireEvent.EventType.IdentifierType = UAIdentifierType_Numeric;
	brsstrcpy((UDINT)&fbUaSrv_FireEvent.EventType.Identifier, (UDINT)&"11436"); // ProgressEventType

	//Parametrieren der anwenderseitigen Felder
	UINT nFieldIndex = 0;
	brsstrcpy((UDINT)&Fields.FieldCfg[nFieldIndex].BrowsePath, (UDINT)&"/Message");
	brsstrcpy((UDINT)&Fields.FieldCfg[nFieldIndex].Variable, (UDINT)&"::SrvEvntC:Fields.Message");
	nFieldIndex += 1;
	brsstrcpy((UDINT)&Fields.FieldCfg[nFieldIndex].BrowsePath, (UDINT)&"/Severity");
	brsstrcpy((UDINT)&Fields.FieldCfg[nFieldIndex].Variable, (UDINT)&"::SrvEvntC:Fields.nSeverity");
	nFieldIndex += 1;
	brsstrcpy((UDINT)&Fields.FieldCfg[nFieldIndex].BrowsePath, (UDINT)&"/Context");
	brsstrcpy((UDINT)&Fields.FieldCfg[nFieldIndex].Variable, (UDINT)&"::SrvEvntC:Fields.Context"); // Hier könnte auch eine Variable eines anderen Standard-Datentyps angebunden werden
	nFieldIndex += 1;
	brsstrcpy((UDINT)&Fields.FieldCfg[nFieldIndex].BrowsePath, (UDINT)&"/Progress");
	brsstrcpy((UDINT)&Fields.FieldCfg[nFieldIndex].Variable, (UDINT)&"::SrvEvntC:Fields.nProgress");
	// Die Felder 'EventId', 'EventType', 'LocalTime', 'ReceiveTime', 'SourceName', 'SourceNode' und 'Time'
	// werden nicht übergeben und daher automatisch vom Betriebssystem besetzt

	fbUaSrv_FireEvent.EventFieldCount = nFieldIndex + 1;
	fbUaSrv_FireEvent.EventFields = (UaSrv_FireEventFieldType*)&Fields.FieldCfg;

	// Sonstige Initialisierung
	fbDelay.PT = 5000; // = 5s
	bSuspendTimer = 0;

	// Initialisierung der Schrittkette
	Step.eStepNr = eSTEP_INIT;

}

void _CYCLIC Cyclic(void)
{
	// Schrittkette
	switch(Step.eStepNr)
	{
		case eSTEP_INIT:
			// Start
			nNamespaceIndexBrPv = 0;
			bFire = 0;
			Step.eStepNr = eSTEP_GET_NS_ORG;
			break;

		case eSTEP_GET_NS_ORG:
			// Ermitteln des Namespace-Index für Foundation-Adressbereich am B&R-Server
			fbUaSrv_GetNamespaceIndex.Execute = 1;
			brsstrcpy((UDINT)&fbUaSrv_GetNamespaceIndex.NamespaceUri, (UDINT)&"http://opcfoundation.org/UA/");
			if(fbUaSrv_GetNamespaceIndex.Done == 1)
			{
				fbUaSrv_GetNamespaceIndex.Execute = 0;
				nNamespaceIndexFoundation = fbUaSrv_GetNamespaceIndex.NamespaceIndex;
				fbUaSrv_FireEvent.EventType.NamespaceIndex = nNamespaceIndexFoundation;
				Step.eStepNr = eSTEP_GET_NS_BR_PV;
			}
			else if(fbUaSrv_GetNamespaceIndex.Error == 1)
			{
				fbUaSrv_GetNamespaceIndex.Execute = 0;
				Step.eErrorStep = eSTEP_GET_NS_ORG;
				Step.nErrorId = fbUaSrv_GetNamespaceIndex.ErrorID;
				Step.nFieldIndex = -1;
				Step.eStepNr = eSTEP_GET_NS_ORG;
			}
			break;

		case eSTEP_GET_NS_BR_PV:
			// Ermitteln des Namespace-Index für PV-Adressbereich am B&R-Server
			fbUaSrv_GetNamespaceIndex.Execute = 1;
			brsstrcpy((UDINT)&fbUaSrv_GetNamespaceIndex.NamespaceUri, (UDINT)&"http://br-automation.com/OpcUa/PLC/PV/");
			if(fbUaSrv_GetNamespaceIndex.Done == 1)
			{
				fbUaSrv_GetNamespaceIndex.Execute = 0;
				nNamespaceIndexBrPv = fbUaSrv_GetNamespaceIndex.NamespaceIndex;
				Step.eStepNr = eSTEP_DELAY;
			}
			else if(fbUaSrv_GetNamespaceIndex.Error == 1)
			{
				fbUaSrv_GetNamespaceIndex.Execute = 0;
				Step.eErrorStep = eSTEP_GET_NS_BR_PV;
				Step.nErrorId = fbUaSrv_GetNamespaceIndex.ErrorID;
				Step.nFieldIndex = -1;
				Step.eStepNr = eSTEP_GET_NS_BR_PV;
			}
			break;

		case eSTEP_DELAY:
			// Warten, bis Event gefeuert werden soll
			fbDelay.IN = !bSuspendTimer;
			if(fbDelay.Q == 1)
			{
				fbDelay.IN = 0;
				bFire = 1;
			}
			if(bFire == 1)
			{
				bFire = 0;
				Step.eStepNr = eSTEP_SET_FIELD_VALUES;
			}
			break;

		case eSTEP_SET_FIELD_VALUES:
			// Fortschritt erhöhen
			Fields.nProgress += 1;
			if(Fields.nProgress > 100)
			{
				Fields.nProgress = 0;
			}
			// Besetzen der anwenderseitigen Felder. Sie können bei jedem Feuern anders besetzt werden.
			brsstrcpy((UDINT)&Fields.Message.Locale, (UDINT)&"en");
			brsstrcpy((UDINT)&Fields.Message.Text, (UDINT)&"Progress at Task 'SrvEvntC' has changed to '");
			brsitoa((DINT)Fields.nProgress, (UDINT)&sHelp);
			brsstrcat((UDINT)&Fields.Message.Text, (UDINT)&sHelp);
			brsstrcat((UDINT)&Fields.Message.Text, (UDINT)&"'.");
			Fields.nSeverity = (UINT)BrbGetRandomUdint(1, 500);
			Fields.Context.nUsint = (USINT)BrbGetRandomUdint(0,255);
			Fields.Context.rReal = BrbGetRandomPercent();
			BrbUsintToHex(Fields.Context.nUsint, Fields.Context.sString, sizeof(Fields.Context.sString), 0);
			Step.eStepNr = eSTEP_FIRE;
			break;

		case eSTEP_FIRE:
			fbUaSrv_FireEvent.Execute = 1;
			if(fbUaSrv_FireEvent.Done == 1)
			{
				fbUaSrv_FireEvent.Execute = 0;
				Step.eStepNr = eSTEP_DELAY;
			}
			else if(fbUaSrv_FireEvent.Error == 1)
			{
				fbUaSrv_FireEvent.Execute = 0;
				if(fbUaSrv_FireEvent.ErrorID > 0)
				{
					Step.eErrorStep = eSTEP_FIRE;
					Step.nErrorId = fbUaSrv_FireEvent.ErrorID;
					Step.nFieldIndex = -1;
				}
				else
				{
					// Fehler in einem der Fields
					for(nFieldIndex=0; nFieldIndex<fbUaSrv_FireEvent.EventFieldCount; nFieldIndex++)
					{
						if(Fields.FieldCfg[nFieldIndex].ErrorID > 0)
						{
							Step.eErrorStep = eSTEP_FIRE;
							Step.nErrorId = Fields.FieldCfg[nFieldIndex].ErrorID;
							Step.nFieldIndex = (INT)nFieldIndex;
						}
					}
				}
				Step.eStepNr = eSTEP_DELAY;
			}
			break;

	}

	// Aufruf des FB's
	UaSrv_GetNamespaceIndex(&fbUaSrv_GetNamespaceIndex);
	TON(&fbDelay);
	UaSrv_FireEvent(&fbUaSrv_FireEvent);

}

void _EXIT Exit(void)
{
}

// NOLINTEND(readability-*, bugprone-easily-swappable-parameters, bugprone-branch-clone, clang-diagnostic-invalid-utf8, clang-diagnostic-invalid-source-encoding, clang-diagnostic-pointer-arith, clang-diagnostic-strict-prototypes, clang-diagnostic-shadow, clang-diagnostic-bad-function-cast, clang-analyzer-security.insecureAPI.*, hicpp-uppercase-literal-suffix, hicpp-function-size, cppcoreguidelines-*, performance-*)
```

#### SrvEvntC.typ - Local data types
```iecst
TYPE
	Step_TYP : 	STRUCT
		eStepNr : Steps_ENUM;
		eErrorStep : Steps_ENUM;
		nErrorId : DWORD;
		nFieldIndex : INT;
	END_STRUCT;
	Steps_ENUM :
		(
		eSTEP_INIT,
		eSTEP_GET_NS_ORG,
		eSTEP_GET_NS_BR_PV,
		eSTEP_DELAY,
		eSTEP_SET_FIELD_VALUES,
		eSTEP_FIRE
		);
	Fields_TYP : 	STRUCT
		Message : UALocalizedText;
		nSeverity : UINT;
		Context : EventFieldContext_TYP;
		nProgress : UINT;
		FieldCfg : ARRAY[0..nFIELD_INDEX_MAX]OF UaSrv_FireEventFieldType;
	END_STRUCT;
END_TYPE
```

#### SrvEvntC.var - Local variables
```iecst
VAR
	Step : Step_TYP;
	bFire : BOOL;
	bSuspendTimer : BOOL;
	fbDelay : TON;
END_VAR
VAR CONSTANT
	nFIELD_INDEX_MAX : UINT := 4;
END_VAR
VAR
	nFieldIndex : UINT;
	Fields : Fields_TYP;
	fbUaSrv_GetNamespaceIndex : UaSrv_GetNamespaceIndex;
	nNamespaceIndexFoundation : UINT;
	nNamespaceIndexBrPv : UINT;
	sHelp : STRING[80];
	fbUaSrv_FireEvent : UaSrv_FireEvent;
END_VAR
```

### Package Logical/Tasks/ServerEvents/SrvEvntST - Event-Aufruf im Server in ST

### Program Logical/Tasks/ServerEvents/SrvEvntST/SrvEvntST (IEC) - Event-Aufruf im Server in ST

#### Main.st - Init, cyclic, exit code
```iecst
PROGRAM _INIT
	// Ablöschen der Funktionsblöcke und Strukturen
	brsmemset(ADR(fbUaSrv_GetNamespaceIndex), 0, SIZEOF(fbUaSrv_GetNamespaceIndex));
	brsmemset(ADR(fbUaSrv_FireEvent), 0, SIZEOF(fbUaSrv_FireEvent));
	brsmemset(ADR(Fields), 0, SIZEOF(Fields));

	// Setzen des Events 'ProgressEventType'
	fbUaSrv_FireEvent.EventType.NamespaceIndex := 0; // Wird in der Schrittkette ermittelt
	fbUaSrv_FireEvent.EventType.IdentifierType := UAIdentifierType_Numeric;
	fbUaSrv_FireEvent.EventType.Identifier := '11436'; // ProgressEventType

	//Parametrieren der anwenderseitigen Felder
	nFieldIndex := 0;
	Fields.FieldCfg[nFieldIndex].BrowsePath := '/Message';
	Fields.FieldCfg[nFieldIndex].Variable := '::SrvEvntST:Fields.Message';
	nFieldIndex := nFieldIndex + 1;
	Fields.FieldCfg[nFieldIndex].BrowsePath := '/Severity';
	Fields.FieldCfg[nFieldIndex].Variable := '::SrvEvntST:Fields.nSeverity';
	nFieldIndex := nFieldIndex + 1;
	Fields.FieldCfg[nFieldIndex].BrowsePath := '/Context';
	Fields.FieldCfg[nFieldIndex].Variable := '::SrvEvntST:Fields.Context'; // Hier könnte auch eine Variable eines anderen Standard-Datentyps angebunden werden
	nFieldIndex := nFieldIndex + 1;
	Fields.FieldCfg[nFieldIndex].BrowsePath := '/Progress';
	Fields.FieldCfg[nFieldIndex].Variable := '::SrvEvntST:Fields.nProgress';
	// Die Felder 'EventId', 'EventType', 'LocalTime', 'ReceiveTime', 'SourceName', 'SourceNode' und 'Time'
	// werden nicht übergeben und daher automatisch vom Betriebssystem besetzt.

	fbUaSrv_FireEvent.EventFieldCount := nFieldIndex + 1;

	// Sonstige Initialisierung
	fbDelay.PT := t#5s;
	bSuspendTimer := 0;

	// Initialisierung der Schrittkette
	Step.eStepNr := eSTEP_INIT;

END_PROGRAM

PROGRAM _CYCLIC
	// Schrittkette
	CASE Step.eStepNr OF
		eSTEP_INIT:
			// Start
			nNamespaceIndexBrPv := 0;
			bFire := 0;
			Step.eStepNr := eSTEP_GET_NS_ORG;

		eSTEP_GET_NS_ORG:
			// Ermitteln des Namespace-Index für Foundation-Adressbereich am B&R-Server
			fbUaSrv_GetNamespaceIndex.Execute := 1;
			fbUaSrv_GetNamespaceIndex.NamespaceUri := 'http://opcfoundation.org/UA/';
			IF fbUaSrv_GetNamespaceIndex.Done = 1 THEN
				fbUaSrv_GetNamespaceIndex.Execute := 0;
				nNamespaceIndexFoundation := fbUaSrv_GetNamespaceIndex.NamespaceIndex;
				fbUaSrv_FireEvent.EventType.NamespaceIndex := nNamespaceIndexFoundation;
				Step.eStepNr := eSTEP_GET_NS_BR_PV;
			ELSIF fbUaSrv_GetNamespaceIndex.Error = 1 THEN
				fbUaSrv_GetNamespaceIndex.Execute := 0;
				Step.eErrorStep := eSTEP_GET_NS_ORG;
				Step.nErrorId := fbUaSrv_GetNamespaceIndex.ErrorID;
				Step.nFieldIndex := -1;
				Step.eStepNr := eSTEP_GET_NS_ORG;
			END_IF

		eSTEP_GET_NS_BR_PV:
			// Ermitteln des Namespace-Index für PV-Adressbereich am B&R-Server
			fbUaSrv_GetNamespaceIndex.Execute := 1;
			fbUaSrv_GetNamespaceIndex.NamespaceUri := 'http://br-automation.com/OpcUa/PLC/PV/';
			IF fbUaSrv_GetNamespaceIndex.Done = 1 THEN
				fbUaSrv_GetNamespaceIndex.Execute := 0;
				nNamespaceIndexBrPv := fbUaSrv_GetNamespaceIndex.NamespaceIndex;
				Step.eStepNr := eSTEP_DELAY;
			ELSIF fbUaSrv_GetNamespaceIndex.Error = 1 THEN
				fbUaSrv_GetNamespaceIndex.Execute := 0;
				Step.eErrorStep := eSTEP_GET_NS_BR_PV;
				Step.nErrorId := fbUaSrv_GetNamespaceIndex.ErrorID;
				Step.nFieldIndex := -1;
				Step.eStepNr := eSTEP_GET_NS_BR_PV;
			END_IF

		eSTEP_DELAY:
			// Warten, bis Event gefeuert werden soll
			fbDelay.IN := NOT(bSuspendTimer);
			IF fbDelay.Q = 1 THEN
				fbDelay.IN := 0;
				bFire := 1;
			END_IF
			IF bFire = 1 THEN
				bFire := 0;
				Step.eStepNr := eSTEP_SET_FIELD_VALUES;
			END_IF

		eSTEP_SET_FIELD_VALUES:
			// Fortschritt erhöhen
			Fields.nProgress := Fields.nProgress + 1;
			IF Fields.nProgress > 100 THEN
				Fields.nProgress := 0;
			END_IF
			// Besetzen der anwenderseitigen Felder. Sie können bei jedem Feuern anders besetzt werden.
			Fields.Message.Locale := 'en';
			brsstrcpy(ADR(Fields.Message.Text), ADR('Progress at Task $'SrvEvntST$' has changed to $''));
			brsitoa(UINT_TO_DINT(Fields.nProgress), ADR(sHelp));
			brsstrcat(ADR(Fields.Message.Text), ADR(sHelp));
			brsstrcat(ADR(Fields.Message.Text), ADR('$'.'));
			Fields.nSeverity := UDINT_TO_UINT(BrbGetRandomUdint(1, 500));
			Fields.Context.nUsint := DINT_TO_USINT(BrbGetRandomDint(0,255));
			Fields.Context.rReal := BrbGetRandomPercent();
			BrbUsintToHex(Fields.Context.nUsint, Fields.Context.sString, SIZEOF(Fields.Context.sString), 0);
			Step.eStepNr := eSTEP_FIRE;

		eSTEP_FIRE:
			fbUaSrv_FireEvent.Execute := 1;
			IF fbUaSrv_FireEvent.Done = 1 THEN
				fbUaSrv_FireEvent.Execute := 0;
				Step.eStepNr := eSTEP_DELAY;
			ELSIF fbUaSrv_FireEvent.Error = 1 THEN
				fbUaSrv_FireEvent.Execute := 0;
				IF fbUaSrv_FireEvent.ErrorID > 0 THEN
					Step.eErrorStep := eSTEP_FIRE;
					Step.nErrorId := fbUaSrv_FireEvent.ErrorID;
					Step.nFieldIndex := -1;
				ELSE
					// Fehler in einem der Fields
					FOR nFieldIndex := 0 TO fbUaSrv_FireEvent.EventFieldCount DO
						IF Fields.FieldCfg[nFieldIndex].ErrorID > 0 THEN
							Step.eErrorStep := eSTEP_FIRE;
							Step.nErrorId := Fields.FieldCfg[nFieldIndex].ErrorID;
							Step.nFieldIndex := nFieldIndex;
						END_IF
					END_FOR
				END_IF
				Step.eStepNr := eSTEP_DELAY;
			END_IF

	END_CASE

		// Aufruf des FB's
		fbUaSrv_GetNamespaceIndex();
		fbDelay();
		fbUaSrv_FireEvent(EventFields := Fields.FieldCfg[0]);

END_PROGRAM

PROGRAM _EXIT
END_PROGRAM
```

### Package Logical/Tasks/Clients - Clients in verschiedenen Sprachen

### ReadMe.txt
```
Unter Verwendung der Bibliothek 'AsOpcUac' ist hier das Beispiel eines Clients implementiert.

Allgemeine Konfiguration:
	Der Client baut automatisch nach dem Hochlauf der Sps die Verbindung zum Server auf. Die Variable 'bStartClient'
	ist im Init auf '1' gesetzt. Will man den Client nicht automatisch starten, kann diese Variable im Init auf '0' und
	dann im Watch auf '1' gesetzt werden.
	Verbunden wird auf den eigenen Server. Durch Änderung der Parameter kann aber auch auf einen externen Server verbunden
	werden.

	Der Ablauf sieht wie folgt aus:
		1. Aufbauen der Verbindung
		2. Ermitteln des NamespaceIndex für den Namespace der Foundation "http://opcfoundation.org/UA/"
		3. Ermitteln des NamespaceIndex für den Namespace von B&R-Variablen "http://br-automation.com/OpcUa/PLC/PV/"
		4. Anlegen einer Subscription für Variablen
		5. Ermitteln der NodeHandles für die Subscription
		6. Hinzufügen der MonitorItems
		7. Schleife auf 4. Wenn alle Var-Subscriptions angelegt sind, wird auf Punkt 8. gesprungen
		8. Anlegen einer Subscription für Events
		9. Ermitteln des NodeHandles für den EventNotifier-Knoten ns=0;i=2253 (Root/Objects/Server)
		10. Hinzufügen des EventItems mit den zu sendenden Feldern
		11. Ermitteln der NodeHandles für Read
		12. Ermitteln der NodeHandles für Write
		13. Ermitteln der Handles für Methoden
		14. Verbindungs-Abbruch prüfen
		15. Alle 1000ms wird zu 16 gesprungen
		16. Lesen der Read-Werte
		17. Schreiben der Write-Werte
		18. Aufruf der Methode 'Calculate'
		19. Sprung auf 14.

	Variablen-Subscriptions:
		Es werden 3 Subscriptions mit je 4 MonitoredItems angelegt. Die Parameter der Subscriptions sind wie folgt vergeben:
		SubVar[0]:		PublishingInterval: 500ms					Priority: 200
		SubVar[1]:		PublishingInterval: 1000ms				Priority: 100
		SubVar[2]:		PublishingInterval: 2000ms				Priority: 50

		Im Beispiel für AS4.1 wird noch der FB 'UA_MonitoredItemAdd' verwendet.
		Ab AS4.2 ist der FB 'UA_MonitoredItemAddList' verfügbar, der hier verwendet wird.
		Folgendes muss beachtet werden: Wenn der Parameter 'QueueSize' eines MonitoredItems größer als '0' gesetzt wird,
		MUSS für diese Subscription auch der FB 'UA_MonitoredItemOperateList' ZYKLISCH aufgerufen werden, sonst werden
		keine Werte auf die Variablen geschrieben!
		In diesem Beispiel ist QueueSize immer '0', so dass es auch ohne Operate funktioniert.
		Da diese Informationen in diesem Beispiel nicht benötigt werden, werden für die IN/OUT 'ValuesChanged',
		'RemainingValueCount', 'TimeStamps' und	'NodeQualityIds' des FB 'UA_MonitoredItemAddList' in jeder Subscription
		diesselben Arrays referenziert. Sollten diese Werte benötigt werden, so müssten	sie auf verschiedene Arrays
		gelegt werden.
		Abonniert werden alle Standard-Datentypen der Struktur 'ServerData::VarsLocal.ReadOnly'. Das INT-Array	wird nicht
		abonniert. Die empfangenen Werte werden in die lokale Struktur 'ClientXXX:ClientVarsSubscription' eingetragen.

	Event-Subscription:
		Es wird eine zusätzliche Subscription angelegt, in der nur ein Item hinzugefügt wird. Allerdings handelt es sich
		dabei nicht um ein MonitoredItem (also eine Variable), sondern um ein EventItem, um damit Events zu empfangen.
		Die Abonnierung muss auf einem Knoten erfolgen, dessen Attribut 'EventNotifier' auf '1=SubscribeToEvents' gesetzt
		ist. Damit teilt der Server mit, dass dieser Knoten Events feuern kann. Am OpcUa-Server der B&R-Sps gibt es
		standardmässig nur einen solchen Knoten. Das ist ns=0;i=2253 (Root/Objects/Server). Mit ihm können alle Events des
		Servers abonniert	werden.
		Bei der clientseitigen Abonnierung wird dem Server ein Filter übermittelt, der zwei Einstellungen enthält:
			1. Event-Typ
				Er ist als NodeId aufgelegt und enthält den Knoten, der das zu filternde Event angibt. Im Baum sind die
				möglichen Typen ab 'Root/Types/EventTypes/' zu finden. Wird ein Knoten angegeben, werden dieser
				Typ und alle unterlagerten an den Client gesendet. Wird z.B. der Typ ns=0;i= 2041 (BaseEventType) angegeben,
				werden alle Events geschickt.
				In diesem Beispiel wird der Filter auf ns=0;i=11436 (ProgressEventType) gesetzt, da dieses Event im Task
				'ServerEvents' zyklisch gefeuert wird.

			2. Zu sendende Felder
				Die Felder, die der Server bei jedem Event mitsenden soll, sind als Array aufgelegt. Ein Array-Element enthält
				den relativen Browse-Pfad des Feldes. Besetzt werden muss nur die Struktur 'TargetName', wobei TargetName.Name
				den Namen des Feldes enthält.
				In diesem Beispiel sind folgende Felder angegeben:
					'EventId', 'EventType', 'LocalTime', 'Message', 'ReceiveTime', 'Severity', 'SourceName', 'SourceNode' und
						'Time' aus dem Typen 'BaseEventType'.
					'Context' und 'Progress' aus dem Typen 'ProgressEventType'
				Für jedes dieser angemeldeten Felder muss eine Variable bereitgestellt werden, die vom Stack beim Empfangen
				eines Events mit dem jeweiligen Wert gefüllt werden kann. Dazu wird ein String-Array mit den Namen der Variablen
				übergeben. Die Reihenfolge entspricht der Reihenfolge der Felder. Der Datentyp der Variable muss natürlich dem
				des Feldes entsprechen.

		Um nun das Empfangen eines Events applikativ verarbeiten zu können, muss zyklisch der Baustein 'UA_EventItemOperate'
		aufgerufen werden. Sobald dessen Ausgang 'EventProcessed' auf 1 geht, ist ein neues Event empfangen und die Feld-
		Variablen mit den gesendeten Werten besetzt worden.
		In diesem Beispiel sind die Feld-Variablen in der Struktur 'ReceivedEvent' enthalten.
		Beim Erkennen eines neuen Events werden applikativ zwei Dinge getan. Zum einen wird zu Diagnosezwecken der Zähler
			'ReceivedEvent.nReceivedCount' hochgezählt. Zum anderen wird die als Byte-Array empfangene EventId zu einem
			Hex-String gewandelt, um sie so besser anzeigen zu können.

		Hinweis: Auch Audit-Events können mit diesem Konzept empfangen werden. Der Server sendet Audit-Events aber nur, wenn
			eine verschlüsselte Verbindung aufgebaut ist.
		Hinweis: Weitere Informationen zu Events und Felder siehe ReadMe des Tasks 'ServerEvents'.

	Read:
		Alle 1000ms werden Werte gelesen.
		Gelesen werden von der Struktur 'ServerData:VarsLocal.ReadOnly' jeweils die Elemente 'nUdint', 'nDint' und
		'anInt' (Array) und in die entsprechenden Elemente der lokalen Struktur 'ClientXXX:ClientVarsRead' eingetragen.
		Achtung: Zyklisches Lesen (Polling) sollte niemals in einer Applikation implementiert werden! Stattdessen sollte
		unbedingt Subscription verwendet werden. Dieses Beispiel soll lediglich die Besetzung des FB's veranschaulichen.

	Write:
		Alle 1000ms werden Werte geschrieben.
		Geschrieben werden die oben gelesenen Elemente von der lokalen Struktur 'ClientXXX:ClientVarsRead' auf
		'ServerData::WriteXXX'.

	Method 'Calculate'
		Alle 1000ms wird die Methode aufgerufen.
		Die Eingangs-Argumente werden vor dem Aufruf in der lokalen Struktur 'MethCalculateArgs.In' befüllt.
		Nach dem Aufruf sind die Ausgangs-Argumente in der lokalen Struktur 'MethCalculateArgs.Out' abgelegt.

	NamespaceUri und NamespaceIndex:
		Normalerweise würde die NamespaceUri verwendet, um einen Knoten zu adressieren. Da aber die Übertragung eines
		Texts bei jedem Zugriff zu unperformant wäre, wird bei OpcUa der NamespaceUri in einen ebenso eindeutigen
		NamespaceIndex gewandelt.
		Achtung: Der NamespaceIndex ist nicht statisch und muss folglich nach jedem Verbingungsaufbau mit
		'UA_GetNamespaceIndex' ermittelt werden!
		Jeder Knoten könnte theoretisch in einem anderen Namespace untergebracht sein. Weil beim B&R-Server die Variablen
		aber alle im selben Namespace sind,	wird hier der Index nur einmal ermittelt und für jedes Item verwendet.
		Ab AS4.3 ist die NamespaceUri bei B&R geändert worden:
			AS					Version			NamespaceUri
			<=AS4.2			V1.0				urn:B&R/pv/
			>=As4.3			V2.0				http://br-automation.com/OpcUa/PLC/PV/
		Um kombatibel zu älteren Versionen zu bleiben, kann ab AS4.3 die Modell-Version in der System-
		Konfiguration eingestellt werden.
		Ursache der Änderung: Manche OpcUa-Clients von Fremdherstellern hatten Probleme mit dem '&' im Namespace.

	Verbindungsabbruch:
		Bricht die Verbindung zum Server ab (z.B. durch Abstecken eines Kabels oder Neustart des Servers) und kehrt wieder,
		kann das Betriebssystem automatisch die Verbindung komplett (mit Subscriptions + MonitoredItems) wieder
		restaurieren. Der Task überprüft lediglich, ob die Verbindung wiedergekehrt ist.

	Fehler:
		In der Struktur 'Step' wird der zuletzt aufgetretene Fehler gespeichert sowie der Schritt, in dem der Fehler
		aufgetreten ist, ausserdem optional der	Index der Subscription bzw. des Items.
		Bei manchen Fehlern kann trotzdem weiter gearbeitet werden. Wenn zum Beispiel die Parameter eines MonitoredItems
		falsch sind, können die restlichen trotzdem angelegt werden.
		Auf den Schritt 'eSTEP_PAR_ERROR' wird nur dann gesprungen, wenn ein Fehler auftritt, bei dem die Schrittkette
		aufgrund eines falschen Parameters nicht weitergeführt werden kann. Dieser Parameter muss dann unbedingt berichtigt
		werden, weil sonst der Client nicht arbeitet.

	Server-Diagnose:
		Das Ermitteln von Server-Diagnose-Daten (z.B. wie viele und welche Clients verbunden sind) ist hier nicht implementiert.
		Zwar könnte dies auch hier gemacht werden, da	dazu nur die Abonnierung bestimmter Knoten nötig ist. Da diese aber komplexe
		Datentypen mit dynamischen Arrays haben, welche bequemerweise schon in der Bibliothek "BrbLibUa" vordefiniert sind, ist das
		Beispiel dazu auch im Task 'BrbUa' implementiert. Außerdem können interessante Informationen dazu in der Hilfe der
		Bibliothek nachgelesen werden.
```

### Package Logical/Tasks/Clients/ClientC - Client in ANSI-C

### Program Logical/Tasks/Clients/ClientC/ClientC (ANSIC) - Client in ANSI-C
